Fanuc KAREL source: NC0024.KL

-- PROVISIONAL review KL for V940-1; original PC SHA256 8e9c105c89f582993eda1f05c20954bd7e1a6c4676e7d45d473f33a49910ae2c
-- Incomplete behavior may be omitted. Consult companion uncertainty JSON. Do not deploy.
PROGRAM NC0024
%NOLOCKGROUP
-- UNRESOLVED_LOCAL_POOL 1 cells at code offset 3; source declarations unknown
-- DIRECT_LOCAL_WORD_ACCESS alone does not prove INTEGER, REAL, or BOOLEAN
BEGIN
  -- UNRESOLVED_PC offsets 0-8; opcodes 2B,2C,7B
  -- UNRESOLVED_PC offsets 13-20; opcodes 9D,23
  -- UNRESOLVED_PC offsets 25-42; opcodes 21,40,41,42
  -- UNRESOLVED_PC offsets 47-64; opcodes 21,40,41,42
  -- UNRESOLVED_PC offsets 69-86; opcodes 21,40,41,42
  -- UNRESOLVED_PC offsets 91-121; opcodes 21,9D,52,23,7A,40,41,42
  -- UNRESOLVED_PC offsets 126-150; opcodes 21,2E,52,23,7A,43
  -- UNRESOLVED_PC offsets 155-173; opcodes 21,2E,52,23
  -- UNRESOLVED_PC offsets 178-194; opcodes 7A,40,41,42
  -- UNRESOLVED_PC offsets 199-223; opcodes 21,2E,52,23,7A,43
  -- UNRESOLVED_PC offsets 228-246; opcodes 21,2E,52,23
  -- UNRESOLVED_PC offsets 251-267; opcodes 7A,40,41,42
  -- UNRESOLVED_PC offsets 272-296; opcodes 21,2E,52,23,7A,43
  -- UNRESOLVED_PC offsets 301-319; opcodes 21,2E,52,23
  -- UNRESOLVED_PC offsets 329-333; opcodes 7F
  -- UNRESOLVED_PC offsets 338-342; opcodes 27,AA
  -- UNRESOLVED_PC offsets 347-351; opcodes 7F
END NC0024
